// TIA Portal project "FactoryIO_Template_S7-1200_V16_V16" (V16)
// Vorlageprojekt für das Buch mit Zielsystem S7-1200

(* hardware
DEVICE "S7-1200-Station_1"  S7-1200 Station
   slot 0: "Baugruppenträger_0"  Rack  V1.0
   slot 1: "PLC_1"  CPU 1211C DC/DC/DC  6ES7 211-1AE40-0XB0  V4.1
*)

// ===== PLC "PLC_1"  CPU 1211C DC/DC/DC =====

VAR_GLOBAL   // PLC tag table "Standard-Variablentabelle"
   "Tag_1" AT %A0.0 : Bool;
   "Tag_2" AT %E0.0 : Bool;
   "Tag_3" AT %E0.1 : Bool;
   "start" AT %I10.0 : Bool;
   "conveyor 6" AT %Q10.0 : Bool;
   "stop" AT %I10.1 : Bool;
   "Loop Marker" AT %M0.0 : Bool;
   "Diffuse Sensor 1" AT %I10.2 : Bool;
   "Diffuse Sensor 2" AT %I10.3 : Bool;
   "Diffuse Sensor 3" AT %I10.4 : Bool;
   "conveyor 4" AT %Q10.1 : Bool;
   "conveyor 2" AT %Q10.2 : Bool;
   "pivot arm" AT %Q10.3 : Bool;
   "pivot arm belt" AT %Q10.4 : Bool;
END_VAR

FUNCTION "MHJ-PLC-Lab-Function-S71200" : Void   // FC9000, SCL
{ S7_Optimized_Access := 'TRUE' }
VERSION : 0.1
   VAR_TEMP
      rdTimeReturn : Int;
      outputTime : DTL;
      SyncVal : Byte;
      forVal : Int;
      forVal_2 : Int;
      Value : Byte;
   END_VAR
   VAR CONSTANT
      CompVal : Byte := 16#34;
      Value_01 : Byte := 16#11;
      Value_01_DW : DWord := 16#A165_D992;
      Value_02_DW : DWord := 16#58BE_4401;
   END_VAR
BEGIN

   #Value:=PEEK(area := 16#82,
        dbNumber := 0,
        byteOffset := 511);
   #Value := #Value + 1;

   POKE(area := 16#82,
        dbNumber := 0,
        byteOffset := 511,
        value := #Value);

   POKE(area:=16#81,
        dbNumber:=0,
        byteOffset:=1016,
        value:=#Value_01_DW);
   POKE(area := 16#81,
        dbNumber := 0,
        byteOffset := 1020,
        value := #Value_02_DW);

   POKE(area := 16#81,
        dbNumber := 0,
        byteOffset := 511,
        value := B#16#00);

   FOR #forVal := 0 TO 120 DO
       FOR #forVal_2:=0 TO 10 DO
           #rdTimeReturn:=RD_SYS_T(#outputTime);
           #rdTimeReturn := WR_SYS_T(#outputTime);
           #rdTimeReturn := RD_SYS_T(#outputTime);
           #rdTimeReturn := WR_SYS_T(#outputTime);
       END_FOR;
       #SyncVal:= PEEK(area := 16#81,
                      dbNumber := 0,
                      byteOffset := 511);
       IF #SyncVal = #CompVal THEN
          GOTO M_1;
       END_IF;
   END_FOR;
   RETURN;

   M_1:
   POKE(area := 16#81,
        dbNumber := 0,
        byteOffset := 511,
        value := B#16#0);
END_FUNCTION

ORGANIZATION_BLOCK "Main"   // OB1, LAD, ProgramCycle
TITLE = "Main Program Sweep (Cycle)"
{ S7_Optimized_Access := 'TRUE' }
VERSION : 0.1
   VAR_INPUT
      Initial_Call : Bool;   // Initial call of this OB
      Remanence : Bool;   // =True, if remanent data are available
   END_VAR
BEGIN

REGION Network 1: Konnektierungsbaustein für PLC-Lab
   // Im Netzwerk 1 wird der Konnektierungsbaustein für PLC-Lab aufgerufen.
   // Dieser Aufruf darf nicht entfernt werden!
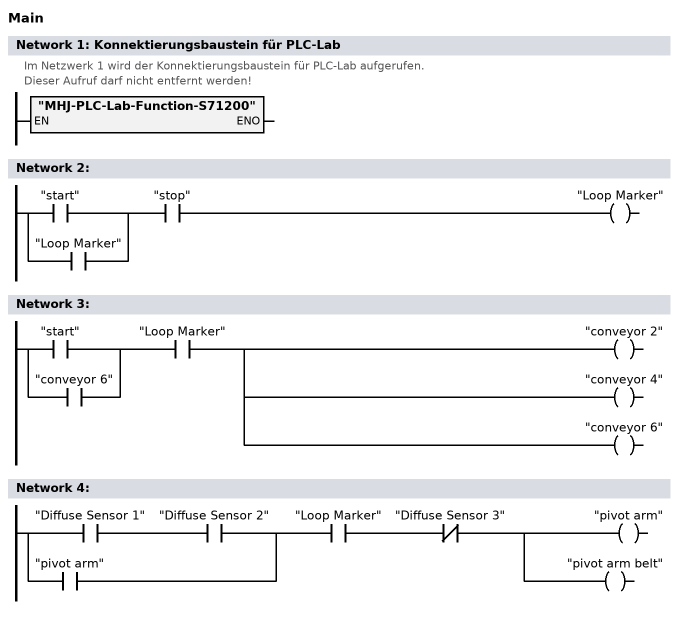
   RUNG wire#powerrail
      "MHJ-PLC-Lab-Function-S71200"()
   END_RUNG
   // the same network as SCL:
   "MHJ-PLC-Lab-Function-S71200"();
END_REGION

REGION Network 2
   RUNG wire#powerrail
      Contact( "start" )
      wire#w1
      Contact( "stop" )
      Coil( "Loop Marker" )
   END_RUNG
   RUNG wire#powerrail
      Contact( "Loop Marker" )
   END_RUNG wire#w1
   // the same network as SCL:
   "Loop Marker" := ("start" OR "Loop Marker") AND "stop";
END_REGION

REGION Network 3
   RUNG wire#powerrail
      Contact( "start" )
      wire#w1
      Contact( "Loop Marker" )
      wire#w2
      Coil( "conveyor 2" )
   END_RUNG
   RUNG wire#powerrail
      Contact( "conveyor 6" )
   END_RUNG wire#w1
   RUNG wire#w2
      Coil( "conveyor 4" )
   END_RUNG
   RUNG wire#w2
      Coil( "conveyor 6" )
   END_RUNG
   // the same network as SCL:
   "conveyor 2" := ("start" OR "conveyor 6") AND "Loop Marker";
   "conveyor 4" := "conveyor 2";
   "conveyor 6" := "conveyor 2";
END_REGION

REGION Network 4
   RUNG wire#powerrail
      Contact( "Diffuse Sensor 1" )
      Contact( "Diffuse Sensor 2" )
      wire#w1
      Contact( "Loop Marker" )
      I_Contact( "Diffuse Sensor 3" )
      wire#w2
      Coil( "pivot arm" )
   END_RUNG
   RUNG wire#powerrail
      Contact( "pivot arm" )
   END_RUNG wire#w1
   RUNG wire#w2
      Coil( "pivot arm belt" )
   END_RUNG
   // the same network as SCL:
   "pivot arm" := (("Diffuse Sensor 1" AND "Diffuse Sensor 2") OR "pivot arm") AND "Loop Marker" AND NOT "Diffuse Sensor 3";
   "pivot arm belt" := "pivot arm";
END_REGION
END_ORGANIZATION_BLOCK